{attribute 'Tc2GvlVarNames'}
VAR_GLOBAL CONSTANT
	maxNumberOfNodes :INT := 22;

	cMSRLIBMaxNumberOfMBusDevices : BYTE := 18;	(*~
				Maximale Anzahl an MBus Geräten, die von der MSRlib unterstützt werden.
				Diese Konstante wird auch für die DP-Historisierung verwendet und muss grösser 6 (Anzahl der Basisdatentypen) sein.
				*)
	cMBUS_MaxData : INT := 40;
	(*cMBUS_MaxTelegrams : INT := 2;
	cMBUS_MaxCom : INT := 1;*)

END_VAR


VAR_GLOBAL

END_VAR

(* stored: Version 1.1.0.1, ProductVersion 3.1.4024.9
   GVL Globale_Variablen: Id {621be69f-e27a-411c-aef3-06a242e2eaec} *)
